GLOBALCONSTANTS DDI (* Global constants *)
  (* Standard: 61499-1 *)
  (* Version 1.0, 2024-02-25, franz *)
  VAR_GLOBAL CONSTANT
    DDI_INTERNAL_DATA_BASE_DDI : UINT := 0; (* 0 - Internal Data Base DDI *)
    DDI_SETPOINT_VOLUME_PER_AREA_APPLICATION_RATE : UINT := 1; (* 1 - Setpoint Volume Per Area Application Rate as *)
    DDI_ACTUAL_VOLUME_PER_AREA_APPLICATION_RATE : UINT := 2; (* 2 - Actual Volume Per Area Application Rate as *)
    DDI_DEFAULT_VOLUME_PER_AREA_APPLICATION_RATE : UINT := 3; (* 3 - Default Volume Per Area Application Rate as *)
    DDI_MINIMUM_VOLUME_PER_AREA_APPLICATION_RATE : UINT := 4; (* 4 - Minimum Volume Per Area Application Rate as *)
    DDI_MAXIMUM_VOLUME_PER_AREA_APPLICATION_RATE : UINT := 5; (* 5 - Maximum Volume Per Area Application Rate as *)
    DDI_SETPOINT_MASS_PER_AREA_APPLICATION_RATE : UINT := 6; (* 6 - Setpoint Mass Per Area Application Rate *)
    DDI_ACTUAL_MASS_PER_AREA_APPLICATION_RATE : UINT := 7; (* 7 - Actual Mass Per Area Application Rate *)
    DDI_DEFAULT_MASS_PER_AREA_APPLICATION_RATE : UINT := 8; (* 8 - Default Mass Per Area Application Rate *)
    DDI_MINIMUM_MASS_PER_AREA_APPLICATION_RATE : UINT := 9; (* 9 - Minimum Mass Per Area Application Rate *)
    DDI_MAXIMUM_MASS_PER_AREA_APPLICATION_RATE : UINT := 10; (* 10 - Maximum Mass Per Area Application Rate *)
    DDI_SETPOINT_COUNT_PER_AREA_APPLICATION_RATE : UINT := 11; (* 11 - Setpoint Count Per Area Application Rate *)
    DDI_ACTUAL_COUNT_PER_AREA_APPLICATION_RATE : UINT := 12; (* 12 - Actual Count Per Area Application Rate *)
    DDI_DEFAULT_COUNT_PER_AREA_APPLICATION_RATE : UINT := 13; (* 13 - Default Count Per Area Application Rate *)
    DDI_MINIMUM_COUNT_PER_AREA_APPLICATION_RATE : UINT := 14; (* 14 - Minimum Count Per Area Application Rate *)
    DDI_MAXIMUM_COUNT_PER_AREA_APPLICATION_RATE : UINT := 15; (* 15 - Maximum Count Per Area Application Rate *)
    DDI_SETPOINT_SPACING_APPLICATION_RATE : UINT := 16; (* 16 - Setpoint Spacing Application Rate *)
    DDI_ACTUAL_SPACING_APPLICATION_RATE : UINT := 17; (* 17 - Actual Spacing Application Rate *)
    DDI_DEFAULT_SPACING_APPLICATION_RATE : UINT := 18; (* 18 - Default Spacing Application Rate *)
    DDI_MINIMUM_SPACING_APPLICATION_RATE : UINT := 19; (* 19 - Minimum Spacing Application Rate *)
    DDI_MAXIMUM_SPACING_APPLICATION_RATE : UINT := 20; (* 20 - Maximum Spacing Application Rate *)
    DDI_SETPOINT_VOLUME_PER_VOLUME_APPLICATION_RATE : UINT := 21; (* 21 - Setpoint Volume Per Volume Application Rate *)
    DDI_ACTUAL_VOLUME_PER_VOLUME_APPLICATION_RATE : UINT := 22; (* 22 - Actual Volume Per Volume Application Rate *)
    DDI_DEFAULT_VOLUME_PER_VOLUME_APPLICATION_RATE : UINT := 23; (* 23 - Default Volume Per Volume Application Rate *)
    DDI_MINIMUM_VOLUME_PER_VOLUME_APPLICATION_RATE : UINT := 24; (* 24 - Minimum Volume Per Volume Application Rate *)
    DDI_MAXIMUM_VOLUME_PER_VOLUME_APPLICATION_RATE : UINT := 25; (* 25 - Maximum Volume Per Volume Application Rate *)
    DDI_SETPOINT_MASS_PER_MASS_APPLICATION_RATE : UINT := 26; (* 26 - Setpoint Mass Per Mass Application Rate *)
    DDI_ACTUAL_MASS_PER_MASS_APPLICATION_RATE : UINT := 27; (* 27 - Actual Mass Per Mass Application Rate *)
    DDI_DEFAULT_MASS_PER_MASS_APPLICATION_RATE : UINT := 28; (* 28 - Default Mass Per Mass Application Rate *)
    DDI_MINIMUM_MASS_PER_MASS_APPLICATION_RATE : UINT := 29; (* 29 - Minimum Mass Per Mass Application Rate *)
    DDI_MAXIMUMMASS_PER_MASS_APPLICATION_RATE : UINT := 30; (* 30 - MaximumMass Per Mass Application Rate *)
    DDI_SETPOINT_VOLUME_PER_MASS_APPLICATION_RATE : UINT := 31; (* 31 - Setpoint Volume Per Mass Application Rate *)
    DDI_ACTUAL_VOLUME_PER_MASS_APPLICATION_RATE : UINT := 32; (* 32 - Actual Volume Per Mass Application Rate *)
    DDI_DEFAULT_VOLUME_PER_MASS_APPLICATION_RATE : UINT := 33; (* 33 - Default Volume Per Mass Application Rate *)
    DDI_MINIMUM_VOLUME_PER_MASS_APPLICATION_RATE : UINT := 34; (* 34 - Minimum Volume Per Mass Application Rate *)
    DDI_MAXIMUM_VOLUME_PER_MASS_APPLICATION_RATE : UINT := 35; (* 35 - Maximum Volume Per Mass Application Rate *)
    DDI_SETPOINT_VOLUME_PER_TIME_APPLICATION_RATE : UINT := 36; (* 36 - Setpoint Volume Per Time Application Rate *)
    DDI_ACTUAL_VOLUME_PER_TIME_APPLICATION_RATE : UINT := 37; (* 37 - Actual Volume Per Time Application Rate *)
    DDI_DEFAULT_VOLUME_PER_TIME_APPLICATION_RATE : UINT := 38; (* 38 - Default Volume Per Time Application Rate *)
    DDI_MINIMUM_VOLUME_PER_TIME_APPLICATION_RATE : UINT := 39; (* 39 - Minimum Volume Per Time Application Rate *)
    DDI_MAXIMUM_VOLUME_PER_TIME_APPLICATION_RATE : UINT := 40; (* 40 - Maximum Volume Per Time Application Rate *)
    DDI_SETPOINT_MASS_PER_TIME_APPLICATION_RATE : UINT := 41; (* 41 - Setpoint Mass Per Time Application Rate *)
    DDI_ACTUAL_MASS_PER_TIME_APPLICATION_RATE : UINT := 42; (* 42 - Actual Mass Per Time Application Rate *)
    DDI_DEFAULT_MASS_PER_TIME_APPLICATION_RATE : UINT := 43; (* 43 - Default Mass Per Time Application Rate *)
    DDI_MINIMUM_MASS_PER_TIME_APPLICATION_RATE : UINT := 44; (* 44 - Minimum Mass Per Time Application Rate *)
    DDI_MAXIMUM_MASS_PER_TIME_APPLICATION_RATE : UINT := 45; (* 45 - Maximum Mass Per Time Application Rate *)
    DDI_SETPOINT_COUNT_PER_TIME_APPLICATION_RATE : UINT := 46; (* 46 - Setpoint Count Per Time Application Rate *)
    DDI_ACTUAL_COUNT_PER_TIME_APPLICATION_RATE : UINT := 47; (* 47 - Actual Count Per Time Application Rate *)
    DDI_DEFAULT_COUNT_PER_TIME_APPLICATION_RATE : UINT := 48; (* 48 - Default Count Per Time Application Rate *)
    DDI_MINIMUM_COUNT_PER_TIME_APPLICATION_RATE : UINT := 49; (* 49 - Minimum Count Per Time Application Rate *)
    DDI_MAXIMUM_COUNT_PER_TIME_APPLICATION_RATE : UINT := 50; (* 50 - Maximum Count Per Time Application Rate *)
    DDI_SETPOINT_TILLAGE_DEPTH : UINT := 51; (* 51 - Setpoint Tillage Depth *)
    DDI_ACTUAL_TILLAGE_DEPTH : UINT := 52; (* 52 - Actual Tillage Depth *)
    DDI_DEFAULT_TILLAGE_DEPTH : UINT := 53; (* 53 - Default Tillage Depth *)
    DDI_MINIMUM_TILLAGE_DEPTH : UINT := 54; (* 54 - Minimum Tillage Depth *)
    DDI_MAXIMUM_TILLAGE_DEPTH : UINT := 55; (* 55 - Maximum Tillage Depth *)
    DDI_SETPOINT_SEEDING_DEPTH : UINT := 56; (* 56 - Setpoint Seeding Depth *)
    DDI_ACTUAL_SEEDING_DEPTH : UINT := 57; (* 57 - Actual Seeding Depth *)
    DDI_DEFAULT_SEEDING_DEPTH : UINT := 58; (* 58 - Default Seeding Depth *)
    DDI_MINIMUM_SEEDING_DEPTH : UINT := 59; (* 59 - Minimum Seeding Depth *)
    DDI_MAXIMUM_SEEDING_DEPTH : UINT := 60; (* 60 - Maximum Seeding Depth *)
    DDI_SETPOINT_WORKING_HEIGHT : UINT := 61; (* 61 - Setpoint Working Height *)
    DDI_ACTUAL_WORKING_HEIGHT : UINT := 62; (* 62 - Actual Working Height *)
    DDI_DEFAULT_WORKING_HEIGHT : UINT := 63; (* 63 - Default Working Height *)
    DDI_MINIMUM_WORKING_HEIGHT : UINT := 64; (* 64 - Minimum Working Height *)
    DDI_MAXIMUM_WORKING_HEIGHT : UINT := 65; (* 65 - Maximum Working Height *)
    DDI_SETPOINT_WORKING_WIDTH : UINT := 66; (* 66 - Setpoint Working Width *)
    DDI_ACTUAL_WORKING_WIDTH : UINT := 67; (* 67 - Actual Working Width *)
    DDI_DEFAULT_WORKING_WIDTH : UINT := 68; (* 68 - Default Working Width *)
    DDI_MINIMUM_WORKING_WIDTH : UINT := 69; (* 69 - Minimum Working Width *)
    DDI_MAXIMUM_WORKING_WIDTH : UINT := 70; (* 70 - Maximum Working Width *)
    DDI_SETPOINT_VOLUME_CONTENT : UINT := 71; (* 71 - Setpoint Volume Content *)
    DDI_ACTUAL_VOLUME_CONTENT : UINT := 72; (* 72 - Actual Volume Content *)
    DDI_MAXIMUM_VOLUME_CONTENT : UINT := 73; (* 73 - Maximum Volume Content *)
    DDI_SETPOINT_MASS_CONTENT : UINT := 74; (* 74 - Setpoint Mass Content *)
    DDI_ACTUAL_MASS_CONTENT : UINT := 75; (* 75 - Actual Mass Content *)
    DDI_MAXIMUM_MASS_CONTENT : UINT := 76; (* 76 - Maximum Mass Content *)
    DDI_SETPOINT_COUNT_CONTENT : UINT := 77; (* 77 - Setpoint Count Content *)
    DDI_ACTUAL_COUNT_CONTENT : UINT := 78; (* 78 - Actual Count Content *)
    DDI_MAXIMUM_COUNT_CONTENT : UINT := 79; (* 79 - Maximum Count Content *)
    DDI_APPLICATION_TOTAL_VOLUME_AS_L : UINT := 80; (* 80 - Application Total Volume as [L] *)
    DDI_APPLICATION_TOTAL_MASS_IN_KG : UINT := 81; (* 81 - Application Total Mass in [kg] *)
    DDI_APPLICATION_TOTAL_COUNT : UINT := 82; (* 82 - Application Total Count *)
    DDI_VOLUME_PER_AREA_YIELD : UINT := 83; (* 83 - Volume Per Area Yield *)
    DDI_MASS_PER_AREA_YIELD : UINT := 84; (* 84 - Mass Per Area Yield *)
    DDI_COUNT_PER_AREA_YIELD : UINT := 85; (* 85 - Count Per Area Yield *)
    DDI_VOLUME_PER_TIME_YIELD : UINT := 86; (* 86 - Volume Per Time Yield *)
    DDI_MASS_PER_TIME_YIELD : UINT := 87; (* 87 - Mass Per Time Yield *)
    DDI_COUNT_PER_TIME_YIELD : UINT := 88; (* 88 - Count Per Time Yield *)
    DDI_YIELD_TOTAL_VOLUME : UINT := 89; (* 89 - Yield Total Volume *)
    DDI_YIELD_TOTAL_MASS : UINT := 90; (* 90 - Yield Total Mass *)
    DDI_YIELD_TOTAL_COUNT : UINT := 91; (* 91 - Yield Total Count *)
    DDI_VOLUME_PER_AREA_CROP_LOSS : UINT := 92; (* 92 - Volume Per Area Crop Loss *)
    DDI_MASS_PER_AREA_CROP_LOSS : UINT := 93; (* 93 - Mass Per Area Crop Loss *)
    DDI_COUNT_PER_AREA_CROP_LOSS : UINT := 94; (* 94 - Count Per Area Crop Loss *)
    DDI_VOLUME_PER_TIME_CROP_LOSS : UINT := 95; (* 95 - Volume Per Time Crop Loss *)
    DDI_MASS_PER_TIME_CROP_LOSS : UINT := 96; (* 96 - Mass Per Time Crop Loss *)
    DDI_COUNT_PER_TIME_CROP_LOSS : UINT := 97; (* 97 - Count Per Time Crop Loss *)
    DDI_PERCENTAGE_CROP_LOSS : UINT := 98; (* 98 - Percentage Crop Loss *)
    DDI_CROP_MOISTURE : UINT := 99; (* 99 - Crop Moisture *)
    DDI_CROP_CONTAMINATION : UINT := 100; (* 100 - Crop Contamination *)
    DDI_SETPOINT_BALE_WIDTH : UINT := 101; (* 101 - Setpoint Bale Width *)
    DDI_ACTUAL_BALE_WIDTH : UINT := 102; (* 102 - Actual Bale Width *)
    DDI_DEFAULT_BALE_WIDTH : UINT := 103; (* 103 - Default Bale Width *)
    DDI_MINIMUM_BALE_WIDTH : UINT := 104; (* 104 - Minimum Bale Width *)
    DDI_MAXIMUM_BALE_WIDTH : UINT := 105; (* 105 - Maximum Bale Width *)
    DDI_SETPOINT_BALE_HEIGHT : UINT := 106; (* 106 - Setpoint Bale Height *)
    DDI_ACTUALBALEHEIGHT : UINT := 107; (* 107 - ActualBaleHeight *)
    DDI_DEFAULT_BALE_HEIGHT : UINT := 108; (* 108 - Default Bale Height *)
    DDI_MINIMUM_BALE_HEIGHT : UINT := 109; (* 109 - Minimum Bale Height *)
    DDI_MAXIMUM_BALE_HEIGHT : UINT := 110; (* 110 - Maximum Bale Height *)
    DDI_SETPOINT_BALE_SIZE : UINT := 111; (* 111 - Setpoint Bale Size *)
    DDI_ACTUAL_BALE_SIZE : UINT := 112; (* 112 - Actual Bale Size *)
    DDI_DEFAULT_BALE_SIZE : UINT := 113; (* 113 - Default Bale Size *)
    DDI_MINIMUM_BALE_SIZE : UINT := 114; (* 114 - Minimum Bale Size *)
    DDI_MAXIMUM_BALE_SIZE : UINT := 115; (* 115 - Maximum Bale Size *)
    DDI_TOTAL_AREA : UINT := 116; (* 116 - Total Area *)
    DDI_EFFECTIVE_TOTAL_DISTANCE : UINT := 117; (* 117 - Effective Total Distance *)
    DDI_INEFFECTIVE_TOTAL_DISTANCE : UINT := 118; (* 118 - Ineffective Total Distance *)
    DDI_EFFECTIVE_TOTAL_TIME : UINT := 119; (* 119 - Effective Total Time *)
    DDI_INEFFECTIVE_TOTAL_TIME : UINT := 120; (* 120 - Ineffective Total Time *)
    DDI_PRODUCT_DENSITY_MASS_PER_VOLUME : UINT := 121; (* 121 - Product Density Mass Per Volume *)
    DDI_PRODUCT_DENSITY_MASS_PERCOUNT : UINT := 122; (* 122 - Product Density Mass PerCount *)
    DDI_PRODUCT_DENSITY_VOLUME_PER_COUNT : UINT := 123; (* 123 - Product Density Volume Per Count *)
    DDI_AUXILIARY_VALVE_SCALING_EXTEND : UINT := 124; (* 124 - Auxiliary Valve Scaling Extend *)
    DDI_AUXILIARY_VALVE_SCALING_RETRACT : UINT := 125; (* 125 - Auxiliary Valve Scaling Retract *)
    DDI_AUXILIARY_VALVE_RAMP_EXTEND_UP : UINT := 126; (* 126 - Auxiliary Valve Ramp Extend Up *)
    DDI_AUXILIARY_VALVE_RAMP_EXTEND_DOWN : UINT := 127; (* 127 - Auxiliary Valve Ramp Extend Down *)
    DDI_AUXILIARY_VALVE_RAMP_RETRACT_UP : UINT := 128; (* 128 - Auxiliary Valve Ramp Retract Up *)
    DDI_AUXILIARY_VALVE_RAMP_RETRACT_DOWN : UINT := 129; (* 129 - Auxiliary Valve Ramp Retract Down *)
    DDI_AUXILIARY_VALVE_FLOAT_THRESHOLD : UINT := 130; (* 130 - Auxiliary Valve Float Threshold *)
    DDI_AUXILIARY_VALVE_PROGRESSIVITY_EXTEND : UINT := 131; (* 131 - Auxiliary Valve Progressivity Extend *)
    DDI_AUXILIARY_VALVE_PROGRESSIVITY_RETRACT : UINT := 132; (* 132 - Auxiliary Valve Progressivity Retract *)
    DDI_AUXILIARY_VALVE_INVERT_PORTS : UINT := 133; (* 133 - Auxiliary Valve Invert Ports *)
    DDI_DEVICE_ELEMENT_OFFSET_X : UINT := 134; (* 134 - Device Element Offset X *)
    DDI_DEVICE_ELEMENT_OFFSET_Y : UINT := 135; (* 135 - Device Element Offset Y *)
    DDI_DEVICE_ELEMENT_OFFSET_Z : UINT := 136; (* 136 - Device Element Offset Z *)
    DDI_DEVICE_VOLUME_CAPACITY : UINT := 137; (* 137 - Device Volume Capacity *)
    DDI_DEVICE_MASS_CAPACITY : UINT := 138; (* 138 - Device Mass Capacity *)
    DDI_DEVICE_COUNT_CAPACITY : UINT := 139; (* 139 - Device Count Capacity *)
    DDI_SETPOINT_PERCENTAGE_APPLICATION_RATE : UINT := 140; (* 140 - Setpoint Percentage Application Rate *)
    DDI_ACTUAL_WORK_STATE : UINT := 141; (* 141 - Actual Work State *)
    DDI_PHYSICAL_SETPOINT_TIME_LATENCY : UINT := 142; (* 142 - Physical Setpoint Time Latency *)
    DDI_PHYSICAL_ACTUAL_VALUE_TIME_LATENCY : UINT := 143; (* 143 - Physical Actual Value Time Latency *)
    DDI_YAW_ANGLE : UINT := 144; (* 144 - Yaw Angle *)
    DDI_ROLL_ANGLE : UINT := 145; (* 145 - Roll Angle *)
    DDI_PITCH_ANGLE : UINT := 146; (* 146 - Pitch Angle *)
    DDI_LOG_COUNT : UINT := 147; (* 147 - Log Count *)
    DDI_TOTAL_FUEL_CONSUMPTION : UINT := 148; (* 148 - Total Fuel Consumption *)
    DDI_INSTANTANEOUS_FUEL_CONSUMPTION_PER_TIME : UINT := 149; (* 149 - Instantaneous Fuel Consumption per Time *)
    DDI_INSTANTANEOUS_FUEL_CONSUMPTION_PER_AREA : UINT := 150; (* 150 - Instantaneous Fuel Consumption per Area *)
    DDI_INSTANTANEOUS_AREA_PER_TIME_CAPACITY : UINT := 151; (* 151 - Instantaneous Area Per Time Capacity *)
    DDI_ACTUAL_NORMALIZED_DIFFERENCE_VEGETATIVE_INDEX_NDVI : UINT := 153; (* 153 - Actual Normalized Difference *)
    DDI_PHYSICAL_OBJECT_LENGTH : UINT := 154; (* 154 - Physical Object Length *)
    DDI_PHYSICAL_OBJECT_WIDTH : UINT := 155; (* 155 - Physical Object Width *)
    DDI_PHYSICAL_OBJECT_HEIGHT : UINT := 156; (* 156 - Physical Object Height *)
    DDI_CONNECTOR_TYPE : UINT := 157; (* 157 - Connector Type *)
    DDI_PRESCRIPTION_CONTROL_STATE : UINT := 158; (* 158 - Prescription Control State *)
    DDI_NUMBER_OF_SUB_UNITS_PER_SECTION : UINT := 159; (* 159 - Number of Sub-Units per Section *)
    DDI_SECTION_CONTROL_STATE : UINT := 160; (* 160 - Section Control State *)
    DDI_ACTUAL_CONDENSED_WORK_STATE_1_16 : UINT := 161; (* 161 - Actual Condensed Work State (1-16) *)
    DDI_ACTUAL_CONDENSED_WORK_STATE_17_32 : UINT := 162; (* 162 - Actual Condensed Work State (17-32) *)
    DDI_ACTUAL_CONDENSED_WORK_STATE_33_48 : UINT := 163; (* 163 - Actual Condensed Work State (33-48) *)
    DDI_ACTUAL_CONDENSED_WORK_STATE_49_64 : UINT := 164; (* 164 - Actual Condensed Work State (49-64) *)
    DDI_ACTUAL_CONDENSED_WORK_STATE_65_80 : UINT := 165; (* 165 - Actual Condensed Work State (65-80) *)
    DDI_ACTUAL_CONDENSED_WORK_STATE_81_96 : UINT := 166; (* 166 - Actual Condensed Work State (81-96) *)
    DDI_ACTUAL_CONDENSED_WORK_STATE_97_112 : UINT := 167; (* 167 - Actual Condensed Work State (97-112) *)
    DDI_ACTUAL_CONDENSED_WORK_STATE_113_128 : UINT := 168; (* 168 - Actual Condensed Work State (113-128) *)
    DDI_ACTUAL_CONDENSED_WORK_STATE_129_144 : UINT := 169; (* 169 - Actual Condensed Work State (129-144) *)
    DDI_ACTUAL_CONDENSED_WORK_STATE_145_160 : UINT := 170; (* 170 - Actual Condensed Work State (145-160) *)
    DDI_ACTUAL_CONDENSED_WORK_STATE_161_176 : UINT := 171; (* 171 - Actual Condensed Work State (161-176) *)
    DDI_ACTUAL_CONDENSED_WORK_STATE_177_192 : UINT := 172; (* 172 - Actual Condensed Work State (177-192) *)
    DDI_ACTUAL_CONDENSED_WORK_STATE_193_208 : UINT := 173; (* 173 - Actual Condensed Work State (193-208) *)
    DDI_ACTUAL_CONDENSED_WORK_STATE_209_224 : UINT := 174; (* 174 - Actual Condensed Work State (209-224) *)
    DDI_ACTUAL_CONDENSED_WORK_STATE_225_240 : UINT := 175; (* 175 - Actual Condensed Work State (225-240) *)
    DDI_ACTUAL_CONDENSED_WORK_STATE_241_256 : UINT := 176; (* 176 - Actual Condensed Work State (241-256) *)
    DDI_ACTUAL_LENGTH_OF_CUT : UINT := 177; (* 177 - Actual length of cut *)
    DDI_ELEMENT_TYPE_INSTANCE : UINT := 178; (* 178 - Element Type Instance *)
    DDI_ACTUAL_CULTURAL_PRACTICE : UINT := 179; (* 179 - Actual Cultural Practice *)
    DDI_DEVICE_REFERENCE_POINT_DRP_TO_GROUND_DISTANCE : UINT := 180; (* 180 - Device Reference Point (DRP) to *)
    DDI_DRY_MASS_PER_AREA_YIELD : UINT := 181; (* 181 - Dry Mass Per Area Yield *)
    DDI_DRY_MASS_PER_TIME_YIELD : UINT := 182; (* 182 - Dry Mass Per Time Yield *)
    DDI_YIELD_TOTAL_DRY_MASS : UINT := 183; (* 183 - Yield Total Dry Mass *)
    DDI_REFERENCE_MOISTURE_FOR_DRY_MASS : UINT := 184; (* 184 - Reference Moisture For Dry Mass *)
    DDI_SEED_COTTON_MASS_PER_AREA_YIELD : UINT := 185; (* 185 - Seed Cotton Mass Per Area Yield *)
    DDI_LINT_COTTON_MASS_PER_AREA_YIELD : UINT := 186; (* 186 - Lint Cotton Mass Per Area Yield *)
    DDI_SEED_COTTON_MASS_PER_TIME_YIELD : UINT := 187; (* 187 - Seed Cotton Mass Per Time Yield *)
    DDI_LINT_COTTON_MASS_PER_TIME_YIELD : UINT := 188; (* 188 - Lint Cotton Mass Per Time Yield *)
    DDI_YIELD_TOTAL_SEED_COTTON_MASS : UINT := 189; (* 189 - Yield Total Seed Cotton Mass *)
    DDI_YIELD_TOTAL_LINT_COTTON_MASS : UINT := 190; (* 190 - Yield Total Lint Cotton Mass *)
    DDI_LINT_TURNOUT_PERCENTAGE : UINT := 191; (* 191 - Lint Turnout Percentage *)
    DDI_AMBIENT_TEMPERATURE : UINT := 192; (* 192 - Ambient temperature *)
    DDI_SETPOINT_PRODUCT_PRESSURE : UINT := 193; (* 193 - Setpoint Product Pressure *)
    DDI_ACTUAL_PRODUCT_PRESSURE : UINT := 194; (* 194 - Actual Product Pressure *)
    DDI_MINIMUM_PRODUCT_PRESSURE : UINT := 195; (* 195 - Minimum Product Pressure *)
    DDI_MAXIMUM_PRODUCT_PRESSURE : UINT := 196; (* 196 - Maximum Product Pressure *)
    DDI_SETPOINT_PUMP_OUTPUT_PRESSURE : UINT := 197; (* 197 - Setpoint Pump Output Pressure *)
    DDI_ACTUAL_PUMP_OUTPUT_PRESSURE : UINT := 198; (* 198 - Actual Pump Output Pressure *)
    DDI_MINIMUM_PUMP_OUTPUT_PRESSURE : UINT := 199; (* 199 - Minimum Pump Output Pressure *)
    DDI_MAXIMUM_PUMP_OUTPUT_PRESSURE : UINT := 200; (* 200 - Maximum Pump Output Pressure *)
    DDI_SETPOINT_TANK_AGITATION_PRESSURE : UINT := 201; (* 201 - Setpoint Tank Agitation Pressure *)
    DDI_ACTUAL_TANK_AGITATION_PRESSURE : UINT := 202; (* 202 - Actual Tank Agitation Pressure *)
    DDI_MINIMUM_TANK_AGITATION_PRESSURE : UINT := 203; (* 203 - Minimum Tank Agitation Pressure *)
    DDI_MAXIMUM_TANK_AGITATION_PRESSURE : UINT := 204; (* 204 - Maximum Tank Agitation Pressure *)
    DDI_SC_SETPOINT_TURN_ON_TIME : UINT := 205; (* 205 - SC Setpoint Turn On Time *)
    DDI_SC_SETPOINT_TURN_OFF_TIME : UINT := 206; (* 206 - SC Setpoint Turn Off Time *)
    DDI_WIND_SPEED : UINT := 207; (* 207 - Wind speed *)
    DDI_WIND_DIRECTION : UINT := 208; (* 208 - Wind direction *)
    DDI_RELATIVE_HUMIDITY : UINT := 209; (* 209 - Relative Humidity *)
    DDI_SKY_CONDITIONS : UINT := 210; (* 210 - Sky conditions *)
    DDI_LAST_BALE_FLAKES_PER_BALE : UINT := 211; (* 211 - Last Bale Flakes per Bale *)
    DDI_LAST_BALE_AVERAGE_MOISTURE : UINT := 212; (* 212 - Last Bale Average Moisture *)
    DDI_LAST_BALE_AVERAGE_STROKES_PER_FLAKE : UINT := 213; (* 213 - Last Bale Average Strokes per Flake *)
    DDI_LIFETIME_BALE_COUNT : UINT := 214; (* 214 - Lifetime Bale Count *)
    DDI_LIFETIME_WORKING_HOURS : UINT := 215; (* 215 - Lifetime Working Hours *)
    DDI_ACTUAL_BALE_HYDRAULIC_PRESSURE : UINT := 216; (* 216 - Actual Bale Hydraulic Pressure *)
    DDI_LAST_BALE_AVERAGE_HYDRAULIC_PRESSURE : UINT := 217; (* 217 - Last Bale Average Hydraulic Pressure *)
    DDI_SETPOINT_BALE_COMPRESSION_PLUNGER_LOAD : UINT := 218; (* 218 - Setpoint Bale Compression Plunger Load *)
    DDI_ACTUAL_BALE_COMPRESSION_PLUNGER_LOAD : UINT := 219; (* 219 - Actual Bale Compression Plunger Load *)
    DDI_LAST_BALE_AVERAGE_BALE_COMPRESSION_PLUNGER_LOAD : UINT := 220; (* 220 - Last Bale Average Bale Compression *)
    DDI_LAST_BALE_APPLIED_PRESERVATIVE : UINT := 221; (* 221 - Last Bale Applied Preservative *)
    DDI_LAST_BALE_TAG_NUMBER : UINT := 222; (* 222 - Last Bale Tag Number *)
    DDI_LAST_BALE_MASS : UINT := 223; (* 223 - Last Bale Mass *)
    DDI_DELTA_T : UINT := 224; (* 224 - Delta T *)
    DDI_SETPOINT_WORKING_LENGTH : UINT := 225; (* 225 - Setpoint Working Length *)
    DDI_ACTUAL_WORKING_LENGTH : UINT := 226; (* 226 - Actual Working Length *)
    DDI_MINIMUM_WORKING_LENGTH : UINT := 227; (* 227 - Minimum Working Length *)
    DDI_MAXIMUM_WORKING_LENGTH : UINT := 228; (* 228 - Maximum Working Length *)
    DDI_ACTUAL_NET_WEIGHT : UINT := 229; (* 229 - Actual Net Weight *)
    DDI_NET_WEIGHT_STATE : UINT := 230; (* 230 - Net Weight State *)
    DDI_SETPOINT_NET_WEIGHT : UINT := 231; (* 231 - Setpoint Net Weight *)
    DDI_ACTUAL_GROSS_WEIGHT : UINT := 232; (* 232 - Actual Gross Weight *)
    DDI_GROSS_WEIGHT_STATE : UINT := 233; (* 233 - Gross Weight State *)
    DDI_MINIMUM_GROSS_WEIGHT : UINT := 234; (* 234 - Minimum Gross Weight *)
    DDI_MAXIMUM_GROSS_WEIGHT : UINT := 235; (* 235 - Maximum Gross Weight *)
    DDI_THRESHER_ENGAGEMENT_TOTAL_TIME : UINT := 236; (* 236 - Thresher Engagement Total Time *)
    DDI_ACTUAL_HEADER_WORKING_HEIGHT_STATUS : UINT := 237; (* 237 - Actual Header Working Height Status *)
    DDI_ACTUAL_HEADER_ROTATIONAL_SPEED_STATUS : UINT := 238; (* 238 - Actual Header Rotational Speed Status *)
    DDI_YIELD_HOLD_STATUS : UINT := 239; (* 239 - Yield Hold Status *)
    DDI_ACTUAL_UNLOADING_SYSTEM_STATUS : UINT := 240; (* 240 - Actual (Un)Loading System Status *)
    DDI_CROP_TEMPERATURE : UINT := 241; (* 241 - Crop Temperature *)
    DDI_SETPOINT_SIEVE_CLEARANCE : UINT := 242; (* 242 - Setpoint Sieve Clearance *)
    DDI_ACTUAL_SIEVE_CLEARANCE : UINT := 243; (* 243 - Actual Sieve Clearance *)
    DDI_MINIMUM_SIEVE_CLEARANCE : UINT := 244; (* 244 - Minimum Sieve Clearance *)
    DDI_MAXIMUM_SIEVE_CLEARANCE : UINT := 245; (* 245 - Maximum Sieve Clearance *)
    DDI_SETPOINT_CHAFFER_CLEARANCE : UINT := 246; (* 246 - Setpoint Chaffer Clearance *)
    DDI_ACTUAL_CHAFFER_CLEARANCE : UINT := 247; (* 247 - Actual Chaffer Clearance *)
    DDI_MINIMUM_CHAFFER_CLEARANCE : UINT := 248; (* 248 - Minimum Chaffer Clearance *)
    DDI_MAXIMUM_CHAFFER_CLEARANCE : UINT := 249; (* 249 - Maximum Chaffer Clearance *)
    DDI_SETPOINT_CONCAVE_CLEARANCE : UINT := 250; (* 250 - Setpoint Concave Clearance *)
    DDI_ACTUAL_CONCAVE_CLEARANCE : UINT := 251; (* 251 - Actual Concave Clearance *)
    DDI_MINIMUM_CONCAVE_CLEARANCE : UINT := 252; (* 252 - Minimum Concave Clearance *)
    DDI_MAXIMUM_CONCAVE_CLEARANCE : UINT := 253; (* 253 - Maximum Concave Clearance *)
    DDI_SETPOINT_SEPARATION_FAN_ROTATIONAL_SPEED : UINT := 254; (* 254 - Setpoint Separation Fan Rotational Speed *)
    DDI_ACTUAL_SEPARATION_FAN_ROTATIONAL_SPEED : UINT := 255; (* 255 - Actual Separation Fan Rotational Speed *)
    DDI_MINIMUM_SEPARATION_FAN_ROTATIONAL_SPEED : UINT := 256; (* 256 - Minimum Separation Fan Rotational Speed *)
    DDI_MAXIMUM_SEPARATION_FAN_ROTATIONAL_SPEED : UINT := 257; (* 257 - Maximum Separation Fan Rotational Speed *)
    DDI_HYDRAULIC_OIL_TEMPERATURE : UINT := 258; (* 258 - Hydraulic Oil Temperature *)
    DDI_YIELD_LAG_IGNORE_TIME : UINT := 259; (* 259 - Yield Lag Ignore Time *)
    DDI_YIELD_LEAD_IGNORE_TIME : UINT := 260; (* 260 - Yield Lead Ignore Time *)
    DDI_AVERAGE_YIELD_MASS_PER_TIME : UINT := 261; (* 261 - Average Yield Mass Per Time *)
    DDI_AVERAGE_CROP_MOISTURE : UINT := 262; (* 262 - Average Crop Moisture *)
    DDI_AVERAGE_YIELD_MASS_PER_AREA : UINT := 263; (* 263 - Average Yield Mass Per Area *)
    DDI_CONNECTOR_PIVOT_X_OFFSET : UINT := 264; (* 264 - Connector Pivot X-Offset *)
    DDI_REMAINING_AREA : UINT := 265; (* 265 - Remaining Area *)
    DDI_LIFETIME_APPLICATION_TOTAL_MASS : UINT := 266; (* 266 - Lifetime Application Total Mass *)
    DDI_LIFETIME_APPLICATION_TOTAL_COUNT : UINT := 267; (* 267 - Lifetime Application Total Count *)
    DDI_LIFETIME_YIELD_TOTAL_VOLUME : UINT := 268; (* 268 - Lifetime Yield Total Volume *)
    DDI_LIFETIME_YIELD_TOTAL_MASS : UINT := 269; (* 269 - Lifetime Yield Total Mass *)
    DDI_LIFETIME_YIELD_TOTAL_COUNT : UINT := 270; (* 270 - Lifetime Yield Total Count *)
    DDI_LIFETIME_TOTAL_AREA : UINT := 271; (* 271 - Lifetime Total Area *)
    DDI_LIFETIME_EFFECTIVE_TOTAL_DISTANCE : UINT := 272; (* 272 - Lifetime Effective Total Distance *)
    DDI_LIFETIME_INEFFECTIVE_TOTAL_DISTANCE : UINT := 273; (* 273 - Lifetime Ineffective Total Distance *)
    DDI_LIFETIME_EFFECTIVE_TOTAL_TIME : UINT := 274; (* 274 - Lifetime Effective Total Time *)
    DDI_LIFETIME_INEFFECTIVE_TOTAL_TIME : UINT := 275; (* 275 - Lifetime Ineffective Total Time *)
    DDI_LIFETIME_FUEL_CONSUMPTION : UINT := 276; (* 276 - Lifetime Fuel Consumption *)
    DDI_LIFETIME_AVERAGE_FUEL_CONSUMPTION_PER_TIME : UINT := 277; (* 277 - Lifetime Average Fuel Consumption per Time *)
    DDI_LIFETIME_AVERAGE_FUEL_CONSUMPTION_PER_AREA : UINT := 278; (* 278 - Lifetime Average Fuel Consumption per Area *)
    DDI_LIFETIME_YIELD_TOTAL_DRY_MASS : UINT := 279; (* 279 - Lifetime Yield Total Dry Mass *)
    DDI_LIFETIME_YIELD_TOTAL_SEED_COTTON_MASS : UINT := 280; (* 280 - Lifetime Yield Total Seed Cotton Mass *)
    DDI_LIFETIME_YIELD_TOTAL_LINT_COTTON_MASS : UINT := 281; (* 281 - Lifetime Yield Total Lint Cotton Mass *)
    DDI_LIFETIME_THRESHING_ENGAGEMENT_TOTAL_TIME : UINT := 282; (* 282 - Lifetime Threshing Engagement Total Time *)
    DDI_PRECUT_TOTAL_COUNT : UINT := 283; (* 283 - Precut Total Count *)
    DDI_UNCUT_TOTAL_COUNT : UINT := 284; (* 284 - Uncut Total Count *)
    DDI_LIFETIME_PRECUT_TOTAL_COUNT : UINT := 285; (* 285 - Lifetime Precut Total Count *)
    DDI_LIFETIME_UNCUT_TOTAL_COUNT : UINT := 286; (* 286 - Lifetime Uncut Total Count *)
    DDI_SETPOINT_PRESCRIPTION_MODE : UINT := 287; (* 287 - Setpoint Prescription Mode *)
    DDI_ACTUAL_PRESCRIPTION_MODE : UINT := 288; (* 288 - Actual Prescription Mode *)
    DDI_SETPOINT_WORK_STATE : UINT := 289; (* 289 - Setpoint Work State *)
    DDI_SETPOINT_CONDENSED_WORK_STATE_1_16 : UINT := 290; (* 290 - Setpoint Condensed Work State (1-16) *)
    DDI_SETPOINT_CONDENSED_WORK_STATE_17_32 : UINT := 291; (* 291 - Setpoint Condensed Work State (17-32) *)
    DDI_SETPOINT_CONDENSED_WORK_STATE_33_48 : UINT := 292; (* 292 - Setpoint Condensed Work State (33-48) *)
    DDI_SETPOINT_CONDENSED_WORK_STATE_49_64 : UINT := 293; (* 293 - Setpoint Condensed Work State (49-64) *)
    DDI_SETPOINT_CONDENSED_WORK_STATE_65_80 : UINT := 294; (* 294 - Setpoint Condensed Work State (65-80) *)
    DDI_SETPOINT_CONDENSED_WORK_STATE_81_96 : UINT := 295; (* 295 - Setpoint Condensed Work State (81-96) *)
    DDI_SETPOINT_CONDENSED_WORK_STATE_97_112 : UINT := 296; (* 296 - Setpoint Condensed Work State (97-112) *)
    DDI_SETPOINT_CONDENSED_WORK_STATE_113_128 : UINT := 297; (* 297 - Setpoint Condensed Work State (113-128) *)
    DDI_SETPOINT_CONDENSED_WORK_STATE_129_144 : UINT := 298; (* 298 - Setpoint Condensed Work State (129-144) *)
    DDI_SETPOINT_CONDENSED_WORK_STATE_145_160 : UINT := 299; (* 299 - Setpoint Condensed Work State (145-160) *)
    DDI_SETPOINT_CONDENSED_WORK_STATE_161_176 : UINT := 300; (* 300 - Setpoint Condensed Work State (161-176) *)
    DDI_SETPOINT_CONDENSED_WORK_STATE_177_192 : UINT := 301; (* 301 - Setpoint Condensed Work State (177-192) *)
    DDI_SETPOINT_CONDENSED_WORK_STATE_193_208 : UINT := 302; (* 302 - Setpoint Condensed Work State (193-208) *)
    DDI_SETPOINT_CONDENSED_WORK_STATE_209_224 : UINT := 303; (* 303 - Setpoint Condensed Work State (209-224) *)
    DDI_SETPOINT_CONDENSED_WORK_STATE_225_240 : UINT := 304; (* 304 - Setpoint Condensed Work State (225-240) *)
    DDI_SETPOINT_CONDENSED_WORK_STATE_241_256 : UINT := 305; (* 305 - Setpoint Condensed Work State (241-256) *)
    DDI_TRUE_ROTATION_POINT_X_OFFSET : UINT := 306; (* 306 - True Rotation Point X-Offset *)
    DDI_TRUE_ROTATION_POINT_Y_OFFSET : UINT := 307; (* 307 - True Rotation Point Y-Offset *)
    DDI_ACTUAL_PERCENTAGE_APPLICATION_RATE : UINT := 308; (* 308 - Actual Percentage Application Rate *)
    DDI_MINIMUM_PERCENTAGE_APPLICATION_RATE : UINT := 309; (* 309 - Minimum Percentage Application Rate *)
    DDI_MAXIMUM_PERCENTAGE_APPLICATION_RATE : UINT := 310; (* 310 - Maximum Percentage Application Rate *)
    DDI_RELATIVE_YIELD_POTENTIAL : UINT := 311; (* 311 - Relative Yield Potential *)
    DDI_MINIMUM_RELATIVE_YIELD_POTENTIAL : UINT := 312; (* 312 - Minimum Relative Yield Potential *)
    DDI_MAXIMUM_RELATIVE_YIELD_POTENTIAL : UINT := 313; (* 313 - Maximum Relative Yield Potential *)
    DDI_ACTUAL_PERCENTAGE_CROP_DRY_MATTER : UINT := 314; (* 314 - Actual Percentage Crop Dry Matter *)
    DDI_AVERAGE_PERCENTAGE_CROP_DRY_MATTER : UINT := 315; (* 315 - Average Percentage Crop Dry Matter *)
    DDI_EFFECTIVE_TOTAL_FUEL_CONSUMPTION : UINT := 316; (* 316 - Effective Total Fuel Consumption *)
    DDI_INEFFECTIVE_TOTAL_FUEL_CONSUMPTION : UINT := 317; (* 317 - Ineffective Total Fuel Consumption *)
    DDI_EFFECTIVE_TOTAL_DIESEL_EXHAUST_FLUID_CONSUMPTION : UINT := 318; (* 318 - Effective Total Diesel Exhaust Fluid *)
    DDI_INEFFECTIVE_TOTAL_DIESEL_EXHAUST_FLUID_CONSUMPTION : UINT := 319; (* 319 - Ineffective Total Diesel Exhaust *)
    DDI_LAST_LOADED_WEIGHT : UINT := 320; (* 320 - Last loaded Weight *)
    DDI_LAST_UNLOADED_WEIGHT : UINT := 321; (* 321 - Last unloaded Weight *)
    DDI_LOAD_IDENTIFICATION_NUMBER : UINT := 322; (* 322 - Load Identification Number *)
    DDI_UNLOAD_IDENTIFICATION_NUMBER : UINT := 323; (* 323 - Unload Identification Number *)
    DDI_CHOPPER_ENGAGEMENT_TOTAL_TIME : UINT := 324; (* 324 - Chopper Engagement Total Time *)
    DDI_LIFETIME_APPLICATION_TOTAL_VOLUME : UINT := 325; (* 325 - Lifetime Application Total Volume *)
    DDI_SETPOINT_HEADER_SPEED : UINT := 326; (* 326 - Setpoint Header Speed *)
    DDI_ACTUAL_HEADER_SPEED : UINT := 327; (* 327 - Actual Header Speed *)
    DDI_MINIMUM_HEADER_SPEED : UINT := 328; (* 328 - Minimum Header Speed *)
    DDI_MAXIMUM_HEADER_SPEED : UINT := 329; (* 329 - Maximum Header Speed *)
    DDI_SETPOINT_CUTTING_DRUM_SPEED : UINT := 330; (* 330 - Setpoint Cutting drum speed *)
    DDI_ACTUAL_CUTTING_DRUM_SPEED : UINT := 331; (* 331 - Actual Cutting drum speed *)
    DDI_MINIMUM_CUTTING_DRUM_SPEED : UINT := 332; (* 332 - Minimum Cutting drum speed *)
    DDI_MAXIMUM_CUTTING_DRUM_SPEED : UINT := 333; (* 333 - Maximum Cutting drum speed *)
    DDI_OPERATING_HOURS_SINCE_LAST_SHARPENING : UINT := 334; (* 334 - Operating Hours Since Last Sharpening *)
    DDI_FRONT_PTO_HOURS : UINT := 335; (* 335 - Front PTO hours *)
    DDI_REAR_PTO_HOURS : UINT := 336; (* 336 - Rear PTO hours *)
    DDI_LIFETIME_FRONT_PTO_HOURS : UINT := 337; (* 337 - Lifetime Front PTO hours *)
    DDI_LIFETIME_REAR_PTO_HOURS : UINT := 338; (* 338 - Lifetime Rear PTO Hours *)
    DDI_EFFECTIVE_TOTAL_LOADING_TIME : UINT := 339; (* 339 - Effective Total Loading Time *)
    DDI_EFFECTIVE_TOTAL_UNLOADING_TIME : UINT := 340; (* 340 - Effective Total Unloading Time *)
    DDI_SETPOINT_GRAIN_KERNEL_CRACKER_GAP : UINT := 341; (* 341 - Setpoint Grain Kernel Cracker Gap *)
    DDI_ACTUAL_GRAIN_KERNEL_CRACKER_GAP : UINT := 342; (* 342 - Actual Grain Kernel Cracker Gap *)
    DDI_MINIMUM_GRAIN_KERNEL_CRACKER_GAP : UINT := 343; (* 343 - Minimum Grain Kernel Cracker Gap *)
    DDI_MAXIMUM_GRAIN_KERNEL_CRACKER_GAP : UINT := 344; (* 344 - Maximum Grain Kernel Cracker Gap *)
    DDI_SETPOINT_SWATHING_WIDTH : UINT := 345; (* 345 - Setpoint Swathing Width *)
    DDI_ACTUAL_SWATHING_WIDTH : UINT := 346; (* 346 - Actual Swathing Width *)
    DDI_MINIMUM_SWATHING_WIDTH : UINT := 347; (* 347 - Minimum Swathing Width *)
    DDI_MAXIMUM_SWATHING_WIDTH : UINT := 348; (* 348 - Maximum Swathing Width *)
    DDI_NOZZLE_DRIFT_REDUCTION : UINT := 349; (* 349 - Nozzle Drift Reduction *)
    DDI_FUNCTION_OR_OPERATION_TECHNIQUE : UINT := 350; (* 350 - Function or Operation Technique *)
    DDI_APPLICATION_TOTAL_VOLUME_IN_ML : UINT := 351; (* 351 - Application Total Volume in [ml] *)
    DDI_APPLICATION_TOTAL_MASS_IN_GRAM_G : UINT := 352; (* 352 - Application Total Mass in gram [g] *)
    DDI_TOTAL_APPLICATION_OF_NITROGEN : UINT := 353; (* 353 - Total Application of Nitrogen *)
    DDI_TOTAL_APPLICATION_OF_AMMONIUM : UINT := 354; (* 354 - Total Application of Ammonium *)
    DDI_TOTAL_APPLICATION_OF_PHOSPHOR : UINT := 355; (* 355 - Total Application of Phosphor *)
    DDI_TOTAL_APPLICATION_OF_POTASSIUM : UINT := 356; (* 356 - Total Application of Potassium *)
    DDI_TOTAL_APPLICATION_OF_DRY_MATTER : UINT := 357; (* 357 - Total Application of Dry Matter *)
    DDI_AVERAGE_DRY_YIELD_MASS_PER_TIME : UINT := 358; (* 358 - Average Dry Yield Mass Per Time *)
    DDI_AVERAGE_DRY_YIELD_MASS_PER_AREA : UINT := 359; (* 359 - Average Dry Yield Mass Per Area *)
    DDI_LAST_BALE_SIZE : UINT := 360; (* 360 - Last Bale Size *)
    DDI_LAST_BALE_DENSITY : UINT := 361; (* 361 - Last Bale Density *)
    DDI_TOTAL_BALE_LENGTH : UINT := 362; (* 362 - Total Bale Length *)
    DDI_LAST_BALE_DRY_MASS : UINT := 363; (* 363 - Last Bale Dry Mass *)
    DDI_ACTUAL_FLAKE_SIZE : UINT := 364; (* 364 - Actual Flake Size *)
    DDI_SETPOINT_DOWNFORCE_PRESSURE : UINT := 365; (* 365 - Setpoint Downforce Pressure *)
    DDI_ACTUAL_DOWNFORCE_PRESSURE : UINT := 366; (* 366 - Actual Downforce Pressure *)
    DDI_CONDENSED_SECTION_OVERRIDE_STATE_1_16 : UINT := 367; (* 367 - Condensed Section Override State (1-16) *)
    DDI_CONDENSED_SECTION_OVERRIDE_STATE_17_32 : UINT := 368; (* 368 - Condensed Section Override State (17-32) *)
    DDI_CONDENSED_SECTION_OVERRIDE_STATE_33_48 : UINT := 369; (* 369 - Condensed Section Override State (33-48) *)
    DDI_CONDENSED_SECTION_OVERRIDE_STATE_49_64 : UINT := 370; (* 370 - Condensed Section Override State (49-64) *)
    DDI_CONDENSED_SECTION_OVERRIDE_STATE_65_80 : UINT := 371; (* 371 - Condensed Section Override State (65-80) *)
    DDI_CONDENSED_SECTION_OVERRIDE_STATE_81_96 : UINT := 372; (* 372 - Condensed Section Override State (81-96) *)
    DDI_CONDENSED_SECTION_OVERRIDE_STATE_97_112 : UINT := 373; (* 373 - Condensed Section Override State (97-112) *)
    DDI_CONDENSED_SECTION_OVERRIDE_STATE_113_128 : UINT := 374; (* 374 - Condensed Section Override State (113-128) *)
    DDI_CONDENSED_SECTION_OVERRIDE_STATE_129_144 : UINT := 375; (* 375 - Condensed Section Override State (129-144) *)
    DDI_CONDENSED_SECTION_OVERRIDE_STATE_145_160 : UINT := 376; (* 376 - Condensed Section Override State (145-160) *)
    DDI_CONDENSED_SECTION_OVERRIDE_STATE_161_176 : UINT := 377; (* 377 - Condensed Section Override State (161-176) *)
    DDI_CONDENSED_SECTION_OVERRIDE_STATE_177_192 : UINT := 378; (* 378 - Condensed Section Override State (177-192) *)
    DDI_CONDENSED_SECTION_OVERRIDE_STATE_193_208 : UINT := 379; (* 379 - Condensed Section Override State (193-208) *)
    DDI_CONDENSED_SECTION_OVERRIDE_STATE_209_224 : UINT := 380; (* 380 - Condensed Section Override State (209-224) *)
    DDI_CONDENSED_SECTION_OVERRIDE_STATE_225_240 : UINT := 381; (* 381 - Condensed Section Override State (225-240) *)
    DDI_CONDENSED_SECTION_OVERRIDE_STATE_241_256 : UINT := 382; (* 382 - Condensed Section Override State (241-256) *)
    DDI_APPARENT_WIND_DIRECTION : UINT := 383; (* 383 - Apparent Wind Direction *)
    DDI_APPARENT_WIND_SPEED : UINT := 384; (* 384 - Apparent Wind Speed *)
    DDI_MSL_ATMOSPHERIC_PRESSURE : UINT := 385; (* 385 - MSL Atmospheric Pressure *)
    DDI_ACTUAL_ATMOSPHERIC_PRESSURE : UINT := 386; (* 386 - Actual Atmospheric Pressure *)
    DDI_TOTAL_REVOLUTIONS_IN_FRACTIONAL_REVOLUTIONS : UINT := 387; (* 387 - Total Revolutions in Fractional *)
    DDI_TOTAL_REVOLUTIONS_IN_COMPLETE_REVOLUTIONS : UINT := 388; (* 388 - Total Revolutions in Complete Revolutions *)
    DDI_SETPOINT_REVOLUTIONS_SPECIFIED_AS_COUNT_PER_TIME : UINT := 389; (* 389 - Setpoint Revolutions specified as *)
    DDI_ACTUAL_REVOLUTIONS_PER_TIME : UINT := 390; (* 390 - Actual Revolutions Per Time *)
    DDI_DEFAULT_REVOLUTIONS_PER_TIME : UINT := 391; (* 391 - Default Revolutions Per Time *)
    DDI_MINIMUM_REVOLUTIONS_PER_TIME : UINT := 392; (* 392 - Minimum Revolutions Per Time *)
    DDI_MAXIMUM_REVOLUTIONS_PER_TIME : UINT := 393; (* 393 - Maximum Revolutions Per Time *)
    DDI_ACTUAL_FUEL_TANK_CONTENT : UINT := 394; (* 394 - Actual Fuel Tank Content *)
    DDI_ACTUAL_DIESEL_EXHAUST_FLUID_TANK_CONTENT : UINT := 395; (* 395 - Actual Diesel Exhaust Fluid Tank Content *)
    DDI_SETPOINT_SPEED : UINT := 396; (* 396 - Setpoint Speed *)
    DDI_ACTUAL_SPEED : UINT := 397; (* 397 - Actual Speed *)
    DDI_MINIMUM_SPEED : UINT := 398; (* 398 - Minimum Speed *)
    DDI_MAXIMUM_SPEED : UINT := 399; (* 399 - Maximum Speed *)
    DDI_SPEED_SOURCE : UINT := 400; (* 400 - Speed Source *)
    DDI_ACTUAL_APPLICATION_OF_NITROGEN : UINT := 401; (* 401 - Actual Application of Nitrogen as [mg/l] *)
    DDI_ACTUAL_APPLICATION_OF_AMMONIUM : UINT := 402; (* 402 - Actual application of Ammonium *)
    DDI_ACTUAL_APPLICATION_OF_PHOSPHOR : UINT := 403; (* 403 - Actual application of Phosphor *)
    DDI_ACTUAL_APPLICATION_OF_POTASSIUM : UINT := 404; (* 404 - Actual application of Potassium *)
    DDI_ACTUAL_APPLICATION_OF_DRY_MATTER : UINT := 405; (* 405 - Actual application of Dry Matter *)
    DDI_ACTUAL_PROTEIN_CONTENT : UINT := 406; (* 406 - Actual Protein Content *)
    DDI_AVERAGE_PROTEIN_CONTENT : UINT := 407; (* 407 - Average Protein Content *)
    DDI_AVERAGE_CROP_CONTAMINATION : UINT := 408; (* 408 - Average Crop Contamination *)
    DDI_TOTAL_DIESEL_EXHAUST_FLUID_CONSUMPTION : UINT := 409; (* 409 - Total Diesel Exhaust Fluid Consumption *)
    DDI_INSTANTANEOUS_DIESEL_EXHAUST_FLUID_CONSUMPTION_PER_TIME : UINT := 410; (* 410 - Instantaneous Diesel Exhaust *)
    DDI_INSTANTANEOUS_DIESEL_EXHAUST_FLUID_CONSUMPTION_PER_AREA : UINT := 411; (* 411 - Instantaneous Diesel Exhaust *)
    DDI_LIFETIME_DIESEL_EXHAUST_FLUID_CONSUMPTION : UINT := 412; (* 412 - Lifetime Diesel Exhaust Fluid Consumption *)
    DDI_LIFETIME_AVERAGE_DIESEL_EXHAUST_FLUID_CONSUMPTION_PER_TIME : UINT := 413; (* 413 - Lifetime Average Diesel *)
    DDI_LIFETIME_AVERAGE_DIESEL_EXHAUST_FLUID_CONSUMPTION_PER_AREA : UINT := 414; (* 414 - Lifetime Average Diesel *)
    DDI_ACTUAL_SEED_SINGULATION_PERCENTAGE : UINT := 415; (* 415 - Actual Seed Singulation Percentage *)
    DDI_AVERAGE_SEED_SINGULATION_PERCENTAGE : UINT := 416; (* 416 - Average Seed Singulation Percentage *)
    DDI_ACTUAL_SEED_SKIP_PERCENTAGE : UINT := 417; (* 417 - Actual Seed Skip Percentage *)
    DDI_AVERAGE_SEED_SKIP_PERCENTAGE : UINT := 418; (* 418 - Average Seed Skip Percentage *)
    DDI_ACTUAL_SEED_MULTIPLE_PERCENTAGE : UINT := 419; (* 419 - Actual Seed Multiple Percentage *)
    DDI_AVERAGE_SEED_MULTIPLE_PERCENTAGE : UINT := 420; (* 420 - Average Seed Multiple Percentage *)
    DDI_ACTUAL_SEED_SPACING_DEVIATION : UINT := 421; (* 421 - Actual Seed Spacing Deviation *)
    DDI_AVERAGE_SEED_SPACING_DEVIATION : UINT := 422; (* 422 - Average Seed Spacing Deviation *)
    DDI_ACTUAL_COEFFICIENT_OF_VARIATION_OF_SEED_SPACING_PERCENTAGE : UINT := 423; (* 423 - Actual Coefficient of *)
    DDI_AVERAGE_COEFFICIENT_OF_VARIATION_OF_SEED_SPACING_PERCENTAGE : UINT := 424; (* 424 - Average Coefficient of *)
    DDI_SETPOINT_MAXIMUM_ALLOWED_SEED_SPACING_DEVIATION : UINT := 425; (* 425 - Setpoint Maximum Allowed Seed Spacing *)
    DDI_SETPOINT_DOWNFORCE_AS_FORCE : UINT := 426; (* 426 - Setpoint Downforce as Force *)
    DDI_ACTUAL_DOWNFORCE_AS_FORCE : UINT := 427; (* 427 - Actual Downforce as Force *)
    DDI_LOADED_TOTAL_MASS : UINT := 428; (* 428 - Loaded Total Mass *)
    DDI_UNLOADED_TOTAL_MASS : UINT := 429; (* 429 - Unloaded Total Mass *)
    DDI_LIFETIME_LOADED_TOTAL_MASS : UINT := 430; (* 430 - Lifetime Loaded Total Mass *)
    DDI_LIFETIME_UNLOADED_TOTAL_MASS : UINT := 431; (* 431 - Lifetime Unloaded Total Mass *)
    DDI_SETPOINT_APPLICATION_RATE_OF_NITROGEN : UINT := 432; (* 432 - Setpoint Application Rate of Nitrogen *)
    DDI_ACTUAL_APPLICATION_RATE_OF_NITROGEN : UINT := 433; (* 433 - Actual Application Rate of Nitrogen *)
    DDI_MINIMUM_APPLICATION_RATE_OF_NITROGEN : UINT := 434; (* 434 - Minimum Application Rate of Nitrogen *)
    DDI_MAXIMUM_APPLICATION_RATE_OF_NITROGEN : UINT := 435; (* 435 - Maximum Application Rate of Nitrogen *)
    DDI_SETPOINT_APPLICATION_RATE_OF_AMMONIUM : UINT := 436; (* 436 - Setpoint Application Rate of Ammonium *)
    DDI_ACTUAL_APPLICATION_RATE_OF_AMMONIUM : UINT := 437; (* 437 - Actual Application Rate of Ammonium *)
    DDI_MINIMUM_APPLICATION_RATE_OF_AMMONIUM : UINT := 438; (* 438 - Minimum Application Rate of Ammonium *)
    DDI_MAXIMUM_APPLICATION_RATE_OF_AMMONIUM : UINT := 439; (* 439 - Maximum Application Rate of Ammonium *)
    DDI_SETPOINT_APPLICATION_RATE_OF_PHOSPHOR : UINT := 440; (* 440 - Setpoint Application Rate of Phosphor *)
    DDI_ACTUAL_APPLICATION_RATE_OF_PHOSPHOR : UINT := 441; (* 441 - Actual Application Rate of Phosphor *)
    DDI_MINIMUM_APPLICATION_RATE_OF_PHOSPHOR : UINT := 442; (* 442 - Minimum Application Rate of Phosphor *)
    DDI_MAXIMUM_APPLICATION_RATE_OF_PHOSPHOR : UINT := 443; (* 443 - Maximum Application Rate of Phosphor *)
    DDI_SETPOINT_APPLICATION_RATE_OF_POTASSIUM : UINT := 444; (* 444 - Setpoint Application Rate of Potassium *)
    DDI_ACTUAL_APPLICATION_RATE_OF_POTASSIUM : UINT := 445; (* 445 - Actual Application Rate of Potassium *)
    DDI_MINIMUM_APPLICATION_RATE_OF_POTASSIUM : UINT := 446; (* 446 - Minimum Application Rate of Potassium *)
    DDI_MAXIMUM_APPLICATION_RATE_OF_POTASSIUM : UINT := 447; (* 447 - Maximum Application Rate of Potassium *)
    DDI_SETPOINT_APPLICATION_RATE_OF_DRY_MATTER : UINT := 448; (* 448 - Setpoint Application Rate of Dry Matter *)
    DDI_ACTUAL_APPLICATION_RATE_OF_DRY_MATTER : UINT := 449; (* 449 - Actual Application Rate of Dry Matter *)
    DDI_MINIMUM_APPLICATION_RATE_OF_DRY_MATTER : UINT := 450; (* 450 - Minimum Application Rate of Dry Matter *)
    DDI_MAXIMUM_APPLICATION_RATE_OF_DRY_MATTER : UINT := 451; (* 451 - Maximum Application Rate of Dry Matter *)
    DDI_LOADED_TOTAL_VOLUME : UINT := 452; (* 452 - Loaded Total Volume *)
    DDI_UNLOADED_TOTAL_VOLUME : UINT := 453; (* 453 - Unloaded Total Volume *)
    DDI_LIFETIME_LOADED_TOTAL_VOLUME : UINT := 454; (* 454 - Lifetime loaded Total Volume *)
    DDI_LIFETIME_UNLOADED_TOTAL_VOLUME : UINT := 455; (* 455 - Lifetime Unloaded Total Volume *)
    DDI_LAST_LOADED_VOLUME : UINT := 456; (* 456 - Last loaded Volume *)
    DDI_LAST_UNLOADED_VOLUME : UINT := 457; (* 457 - Last unloaded Volume *)
    DDI_LOADED_TOTAL_COUNT : UINT := 458; (* 458 - Loaded Total Count *)
    DDI_UNLOADED_TOTAL_COUNT : UINT := 459; (* 459 - Unloaded Total Count *)
    DDI_LIFETIME_LOADED_TOTAL_COUNT : UINT := 460; (* 460 - Lifetime Loaded Total Count *)
    DDI_LIFETIME_UNLOADED_TOTAL_COUNT : UINT := 461; (* 461 - Lifetime Unloaded Total Count *)
    DDI_LAST_LOADED_COUNT : UINT := 462; (* 462 - Last loaded Count *)
    DDI_LAST_UNLOADED_COUNT : UINT := 463; (* 463 - Last unloaded Count *)
    DDI_HAUL_COUNTER : UINT := 464; (* 464 - Haul Counter *)
    DDI_LIFETIME_HAUL_COUNTER : UINT := 465; (* 465 - Lifetime Haul Counter *)
    DDI_ACTUAL_RELATIVE_CONNECTOR_ANGLE : UINT := 466; (* 466 - Actual relative connector angle *)
    DDI_ACTUAL_PERCENTAGE_CONTENT : UINT := 467; (* 467 - Actual Percentage Content *)
    DDI_SOIL_SNOW_FROZEN_CONDTION : UINT := 468; (* 468 - Soil Snow/Frozen Condtion *)
    DDI_ESTIMATED_SOIL_WATER_CONDTION : UINT := 469; (* 469 - Estimated Soil Water Condtion *)
    DDI_SOIL_COMPACTION : UINT := 470; (* 470 - Soil Compaction *)
    DDI_SETPOINT_CULTURAL_PRACTICE : UINT := 471; (* 471 - Setpoint Cultural Practice *)
    DDI_SETPOINT_LENGTH_OF_CUT : UINT := 472; (* 472 - Setpoint Length of Cut *)
    DDI_MINIMUM_LENGTH_OF_CUT : UINT := 473; (* 473 - Minimum length of cut *)
    DDI_MAXIMUM_LENGTH_OF_CUT : UINT := 474; (* 474 - Maximum Length of Cut *)
    DDI_SETPOINT_BALE_HYDRAULIC_PRESSURE : UINT := 475; (* 475 - Setpoint Bale Hydraulic Pressure *)
    DDI_MINIMUM_BALE_HYDRAULIC_PRESSURE : UINT := 476; (* 476 - Minimum Bale Hydraulic Pressure *)
    DDI_MAXIMUM_BALE_HYDRAULIC_PRESSURE : UINT := 477; (* 477 - Maximum Bale Hydraulic Pressure *)
    DDI_SETPOINT_FLAKE_SIZE : UINT := 478; (* 478 - Setpoint Flake Size *)
    DDI_MINIMUM_FLAKE_SIZE : UINT := 479; (* 479 - Minimum Flake Size *)
    DDI_MAXIMUM_FLAKE_SIZE : UINT := 480; (* 480 - Maximum Flake Size *)
    DDI_SETPOINT_NUMBER_OF_SUBBALES : UINT := 481; (* 481 - Setpoint Number of Subbales *)
    DDI_LAST_BALE_NUMBER_OF_SUBBALES : UINT := 482; (* 482 - Last Bale Number of Subbales *)
    DDI_SETPOINT_ENGINE_SPEED : UINT := 483; (* 483 - Setpoint Engine Speed *)
    DDI_ACTUAL_ENGINE_SPEED : UINT := 484; (* 484 - Actual Engine Speed *)
    DDI_MINIMUM_ENGINE_SPEED : UINT := 485; (* 485 - Minimum Engine Speed *)
    DDI_MAXIMUM_ENGINE_SPEED : UINT := 486; (* 486 - Maximum Engine Speed *)
    DDI_DIESEL_EXHAUST_FLUID_TANK_PERCENTAGE_LEVEL : UINT := 488; (* 488 - Diesel Exhaust Fluid Tank Percentage Level *)
    DDI_MAXIMUM_DIESEL_EXHAUST_FLUID_TANK_CONTENT : UINT := 489; (* 489 - Maximum Diesel Exhaust Fluid Tank Content *)
    DDI_MAXIMUM_FUEL_TANK_CONTENT : UINT := 490; (* 490 - Maximum Fuel Tank Content *)
    DDI_FUEL_PERCENTAGE_LEVEL : UINT := 491; (* 491 - Fuel Percentage Level *)
    DDI_TOTAL_ENGINE_HOURS : UINT := 492; (* 492 - Total Engine Hours *)
    DDI_LIFETIME_ENGINE_HOURS : UINT := 493; (* 493 - Lifetime Engine Hours *)
    DDI_LAST_EVENT_PARTNER_ID_BYTE_1_4 : UINT := 494; (* 494 - Last Event Partner ID (Byte 1-4) *)
    DDI_LAST_EVENT_PARTNER_ID_BYTE_5_8 : UINT := 495; (* 495 - Last Event Partner ID (Byte 5-8) *)
    DDI_LAST_EVENT_PARTNER_ID_BYTE_9_12 : UINT := 496; (* 496 - Last Event Partner ID (Byte 9-12) *)
    DDI_LAST_EVENT_PARTNER_ID_BYTE_13_16 : UINT := 497; (* 497 - Last Event Partner ID (Byte 13-16) *)
    DDI_LAST_EVENT_PARTNER_ID_TYPE : UINT := 498; (* 498 - Last Event Partner ID Type *)
    DDI_LAST_EVENT_PARTNER_ID_MANUFACTURER_ID_CODE : UINT := 499; (* 499 - Last Event Partner ID Manufacturer ID Code *)
    DDI_LAST_EVENT_PARTNER_ID_DEVICE_CLASS : UINT := 500; (* 500 - Last Event Partner ID Device Class *)
    DDI_SETPOINT_ENGINE_TORQUE : UINT := 501; (* 501 - Setpoint Engine Torque *)
    DDI_ACTUAL_ENGINE_TORQUE : UINT := 502; (* 502 - Actual Engine Torque *)
    DDI_MINIMUM_ENGINE_TORQUE : UINT := 503; (* 503 - Minimum Engine Torque *)
    DDI_MAXIMUM_ENGINE_TORQUE : UINT := 504; (* 504 - Maximum Engine Torque *)
    DDI_TRAMLINE_CONTROL_LEVEL : UINT := 505; (* 505 - Tramline Control Level *)
    DDI_SETPOINT_TRAMLINE_CONTROL_LEVEL : UINT := 506; (* 506 - Setpoint Tramline Control Level *)
    DDI_TRAMLINE_SEQUENCE_NUMBER : UINT := 507; (* 507 - Tramline Sequence Number *)
    DDI_UNIQUE_A_B_GUIDANCE_REFERENCE_LINE_ID : UINT := 508; (* 508 - Unique A-B Guidance Reference Line ID *)
    DDI_ACTUAL_TRACK_NUMBER : UINT := 509; (* 509 - Actual Track Number *)
    DDI_TRACK_NUMBER_TO_THE_RIGHT : UINT := 510; (* 510 - Track Number to the right *)
    DDI_TRACK_NUMBER_TO_THE_LEFT : UINT := 511; (* 511 - Track Number to the left *)
    DDI_GUIDANCE_LINE_SWATH_WIDTH : UINT := 512; (* 512 - Guidance Line Swath Width *)
    DDI_GUIDANCE_LINE_DEVIATION : UINT := 513; (* 513 - Guidance Line Deviation *)
    DDI_GNSS_QUALITY : UINT := 514; (* 514 - GNSS Quality *)
    DDI_TRAMLINE_CONTROL_STATE : UINT := 515; (* 515 - Tramline Control State *)
    DDI_TRAMLINE_OVERDOSING_RATE : UINT := 516; (* 516 - Tramline Overdosing Rate *)
    DDI_SETPOINT_TRAMLINE_CONDENSED_WORK_STATE_1_16 : UINT := 517; (* 517 - Setpoint Tramline Condensed Work State *)
    DDI_ACTUAL_TRAMLINE_CONDENSED_WORK_STATE_1_16 : UINT := 518; (* 518 - Actual Tramline Condensed Work State (1-16) *)
    DDI_LAST_BALE_LIFETIME_COUNT : UINT := 519; (* 519 - Last Bale Lifetime Count *)
    DDI_ACTUAL_CANOPY_HEIGHT : UINT := 520; (* 520 - Actual Canopy Height *)
    DDI_GNSS_INSTALLATION_TYPE : UINT := 521; (* 521 - GNSS Installation Type *)
    DDI_TWINE_BALE_TOTAL_COUNT : UINT := 522; (* 522 - Twine Bale Total Count *)
    DDI_MESH_BALE_TOTAL_COUNT : UINT := 523; (* 523 - Mesh Bale Total Count *)
    DDI_LIFETIME_TWINE_BALE_TOTAL_COUNT : UINT := 524; (* 524 - Lifetime Twine Bale Total Count *)
    DDI_LIFETIME_MESH_BALE_TOTAL_COUNT : UINT := 525; (* 525 - Lifetime Mesh Bale Total Count *)
    DDI_ACTUAL_COOLING_FLUID_TEMPERATURE : UINT := 526; (* 526 - Actual Cooling Fluid Temperature *)
    DDI_LAST_BALE_CAPACITY : UINT := 528; (* 528 - Last Bale Capacity *)
    DDI_SETPOINT_TILLAGE_DISC_GANG_ANGLE : UINT := 529; (* 529 - Setpoint Tillage Disc Gang Angle *)
    DDI_ACTUAL_TILLAGE_DISC_GANG_ANGLE : UINT := 530; (* 530 - Actual Tillage Disc Gang Angle *)
    DDI_ACTUAL_APPLIED_PRESERVATIVE_PER_YIELD_MASS : UINT := 531; (* 531 - Actual Applied Preservative Per Yield Mass *)
    DDI_SETPOINT_APPLIED_PRESERVATIVE_PER_YIELD_MASS : UINT := 532; (* 532 - Setpoint Applied Preservative Per Yield *)
    DDI_DEFAULT_APPLIED_PRESERVATIVE_PER_YIELD_MASS : UINT := 533; (* 533 - Default Applied Preservative Per Yield *)
    DDI_MINIMUM_APPLIED_PRESERVATIVE_PER_YIELD_MASS : UINT := 534; (* 534 - Minimum Applied Preservative Per Yield *)
    DDI_MAXIMUM_APPLIED_PRESERVATIVE_PER_YIELD_MASS : UINT := 535; (* 535 - Maximum Applied Preservative Per Yield *)
    DDI_TOTAL_APPLIED_PRESERVATIVE : UINT := 536; (* 536 - Total Applied Preservative *)
    DDI_LIFETIME_APPLIED_PRESERVATIVE : UINT := 537; (* 537 - Lifetime Applied Preservative *)
    DDI_AVERAGE_APPLIED_PRESERVATIVE_PER_YIELD_MASS : UINT := 538; (* 538 - Average Applied Preservative Per Yield *)
    DDI_ACTUAL_PRESERVATIVE_TANK_VOLUME : UINT := 539; (* 539 - Actual Preservative Tank Volume *)
    DDI_ACTUAL_PRESERVATIVE_TANK_LEVEL : UINT := 540; (* 540 - Actual Preservative Tank Level *)
    DDI_ACTUAL_PTO_SPEED : UINT := 541; (* 541 - Actual PTO Speed *)
    DDI_SETPOINT_PTO_SPEED : UINT := 542; (* 542 - Setpoint PTO Speed *)
    DDI_DEFAULT_PTO_SPEED : UINT := 543; (* 543 - Default PTO Speed *)
    DDI_MINIMUM_PTO_SPEED : UINT := 544; (* 544 - Minimum PTO Speed *)
    DDI_MAXIMUM_PTO_SPEED : UINT := 545; (* 545 - Maximum PTO Speed *)
    DDI_LIFETIME_CHOPPING_ENGAGEMENT_TOTAL_TIME : UINT := 546; (* 546 - Lifetime Chopping Engagement Total Time *)
    DDI_SETPOINT_BALE_COMPRESSION_PLUNGER_LOAD_N : UINT := 547; (* 547 - Setpoint Bale Compression Plunger Load (N) *)
    DDI_ACTUAL_BALE_COMPRESSION_PLUNGER_LOAD_N : UINT := 548; (* 548 - Actual Bale Compression Plunger Load (N) *)
    DDI_LAST_BALE_AVERAGE_BALE_COMPRESSION_PLUNGER_LOAD_N : UINT := 549; (* 549 - Last Bale Average Bale Compression *)
    DDI_GROUND_COVER : UINT := 550; (* 550 - Ground Cover *)
    DDI_ACTUAL_PTO_TORQUE : UINT := 551; (* 551 - Actual PTO Torque *)
    DDI_SETPOINT_PTO_TORQUE : UINT := 552; (* 552 - Setpoint PTO Torque *)
    DDI_DEFAULT_PTO_TORQUE : UINT := 553; (* 553 - Default PTO Torque *)
    DDI_MINIMUM_PTO_TORQUE : UINT := 554; (* 554 - Minimum PTO Torque *)
    DDI_MAXIMUM_PTO_TORQUE : UINT := 555; (* 555 - Maximum PTO Torque *)
    DDI_PRESENT_WEATHER_CONDITIONS : UINT := 556; (* 556 - Present Weather Conditions *)
    DDI_SETPOINT_ELECTRICAL_CURRENT : UINT := 557; (* 557 - Setpoint Electrical Current *)
    DDI_ACTUAL_ELECTRICAL_CURRENT : UINT := 558; (* 558 - Actual Electrical Current *)
    DDI_MINIMUM_ELECTRICAL_CURRENT : UINT := 559; (* 559 - Minimum Electrical Current *)
    DDI_MAXIMUM_ELECTRICAL_CURRENT : UINT := 560; (* 560 - Maximum Electrical Current *)
    DDI_DEFAULT_ELECTRICAL_CURRENT : UINT := 561; (* 561 - Default Electrical Current *)
    DDI_SETPOINT_VOLTAGE : UINT := 562; (* 562 - Setpoint Voltage *)
    DDI_DEFAULT_VOLTAGE : UINT := 563; (* 563 - Default Voltage *)
    DDI_ACTUAL_VOLTAGE : UINT := 564; (* 564 - Actual Voltage *)
    DDI_MINIMUM_VOLTAGE : UINT := 565; (* 565 - Minimum Voltage *)
    DDI_MAXIMUM_VOLTAGE : UINT := 566; (* 566 - Maximum Voltage *)
    DDI_ACTUAL_ELECTRICAL_RESISTANCE : UINT := 567; (* 567 - Actual Electrical Resistance *)
    DDI_SETPOINT_ELECTRICAL_POWER : UINT := 568; (* 568 - Setpoint Electrical Power *)
    DDI_ACTUAL_ELECTRICAL_POWER : UINT := 569; (* 569 - Actual Electrical Power *)
    DDI_DEFAULT_ELECTRICAL_POWER : UINT := 570; (* 570 - Default Electrical Power *)
    DDI_MAXIMUM_ELECTRICAL_POWER : UINT := 571; (* 571 - Maximum Electrical Power *)
    DDI_MINIMUM_ELECTRICAL_POWER : UINT := 572; (* 572 - Minimum Electrical Power *)
    DDI_TOTAL_ELECTRICAL_ENERGY : UINT := 573; (* 573 - Total Electrical Energy *)
    DDI_SETPOINT_ELECTRICAL_ENERGY_PER_AREA_APPLICATION_RATE : UINT := 574; (* 574 - Setpoint Electrical Energy per *)
    DDI_ACTUAL_ELECTRICAL_ENERGY_PER_AREA_APPLICATION_RATE : UINT := 575; (* 575 - Actual Electrical Energy per Area *)
    DDI_MAXIMUM_ELECTRICAL_ENERGY_PER_AREA_APPLICATION_RATE : UINT := 576; (* 576 - Maximum Electrical Energy per *)
    DDI_MINIMUM_ELECTRICAL_ENERGY_PER_AREA_APPLICATION_RATE : UINT := 577; (* 577 - Minimum Electrical Energy per *)
    DDI_SETPOINT_TEMPERATURE : UINT := 578; (* 578 - Setpoint Temperature *)
    DDI_ACTUAL_TEMPERATURE : UINT := 579; (* 579 - Actual Temperature *)
    DDI_MINIMUM_TEMPERATURE : UINT := 580; (* 580 - Minimum Temperature *)
    DDI_MAXIMUM_TEMPERATURE : UINT := 581; (* 581 - Maximum Temperature *)
    DDI_DEFAULT_TEMPERATURE : UINT := 582; (* 582 - Default Temperature *)
    DDI_SETPOINT_FREQUENCY : UINT := 583; (* 583 - Setpoint Frequency *)
    DDI_ACTUAL_FREQUENCY : UINT := 584; (* 584 - Actual Frequency *)
    DDI_MINIMUM_FREQUENCY : UINT := 585; (* 585 - Minimum Frequency *)
    DDI_MAXIMUM_FREQUENCY : UINT := 586; (* 586 - Maximum Frequency *)
    DDI_PREVIOUS_RAINFALL : UINT := 587; (* 587 - Previous Rainfall *)
    DDI_SETPOINT_VOLUME_PER_AREA_APPLICATION_RATE_BIG : UINT := 588; (* 588 - Setpoint Volume Per Area *)
    DDI_ACTUAL_VOLUME_PER_AREA_APPLICATION_RATE_BIG : UINT := 589; (* 589 - Actual Volume Per Area Application *)
    DDI_MINIMUM_VOLUME_PER_AREA_APPLICATION_RATE_BIG : UINT := 590; (* 590 - Minimum Volume Per Area Application *)
    DDI_MAXIMUM_VOLUME_PER_AREA_APPLICATION_RATE_BIG : UINT := 591; (* 591 - Maximum Volume Per Area Application *)
    DDI_DEFAULT_VOLUME_PER_AREA_APPLICATION_RATE_BIG : UINT := 592; (* 592 - Default Volume Per Area Application *)
    DDI_TRACTION_TYPE : UINT := 593; (* 593 - Traction Type *)
    DDI_STEERING_TYPE : UINT := 594; (* 594 - Steering Type *)
    DDI_MACHINE_MODE : UINT := 595; (* 595 - Machine Mode *)
    DDI_CARGO_AREA_COVER_STATE : UINT := 596; (* 596 - Cargo Area Cover State *)
    DDI_TOTAL_DISTANCE : UINT := 597; (* 597 - Total Distance *)
    DDI_LIFETIME_TOTAL_DISTANCE : UINT := 598; (* 598 - Lifetime Total Distance *)
    DDI_TOTAL_DISTANCE_FIELD : UINT := 599; (* 599 - Total Distance Field *)
    DDI_LIFETIME_TOTAL_DISTANCE_FIELD : UINT := 600; (* 600 - Lifetime Total Distance Field *)
    DDI_TOTAL_DISTANCE_STREET : UINT := 601; (* 601 - Total Distance Street *)
    DDI_LIFETIME_TOTAL_DISTANCE_STREET : UINT := 602; (* 602 - Lifetime Total Distance Street *)
    DDI_ACTUAL_TRAMLINE_CONDENSED_WORK_STATE_17_32 : UINT := 603; (* 603 - Actual Tramline Condensed Work State *)
    DDI_ACTUAL_TRAMLINE_CONDENSED_WORK_STATE_33_48 : UINT := 604; (* 604 - Actual Tramline Condensed Work State *)
    DDI_ACTUAL_TRAMLINE_CONDENSED_WORK_STATE_49_64 : UINT := 605; (* 605 - Actual Tramline Condensed Work State *)
    DDI_ACTUAL_TRAMLINE_CONDENSED_WORK_STATE_65_80 : UINT := 606; (* 606 - Actual Tramline Condensed Work State *)
    DDI_ACTUAL_TRAMLINE_CONDENSED_WORK_STATE_81_96 : UINT := 607; (* 607 - Actual Tramline Condensed Work State *)
    DDI_ACTUAL_TRAMLINE_CONDENSED_WORK_STATE_97_112 : UINT := 608; (* 608 - Actual Tramline Condensed Work State *)
    DDI_ACTUAL_TRAMLINE_CONDENSED_WORK_STATE_113_128 : UINT := 609; (* 609 - Actual Tramline Condensed Work State *)
    DDI_ACTUAL_TRAMLINE_CONDENSED_WORK_STATE_129_144 : UINT := 610; (* 610 - Actual Tramline Condensed Work State *)
    DDI_ACTUAL_TRAMLINE_CONDENSED_WORK_STATE_145_160 : UINT := 611; (* 611 - Actual Tramline Condensed Work State *)
    DDI_ACTUAL_TRAMLINE_CONDENSED_WORK_STATE_161_176 : UINT := 612; (* 612 - Actual Tramline Condensed Work State *)
    DDI_ACTUAL_TRAMLINE_CONDENSED_WORK_STATE_177_192 : UINT := 613; (* 613 - Actual Tramline Condensed Work State *)
    DDI_ACTUAL_TRAMLINE_CONDENSED_WORK_STATE_193_208 : UINT := 614; (* 614 - Actual Tramline Condensed Work State *)
    DDI_ACTUAL_TRAMLINE_CONDENSED_WORK_STATE_209_224 : UINT := 615; (* 615 - Actual Tramline Condensed Work State *)
    DDI_ACTUAL_TRAMLINE_CONDENSED_WORK_STATE_225_240 : UINT := 616; (* 616 - Actual Tramline Condensed Work State *)
    DDI_ACTUAL_TRAMLINE_CONDENSED_WORK_STATE_241_256 : UINT := 617; (* 617 - Actual Tramline Condensed Work State *)
    DDI_SETPOINT_TRAMLINE_CONDENSED_WORK_STATE_17_32 : UINT := 618; (* 618 - Setpoint Tramline Condensed Work State *)
    DDI_SETPOINT_TRAMLINE_CONDENSED_WORK_STATE_33_48 : UINT := 619; (* 619 - Setpoint Tramline Condensed Work State *)
    DDI_SETPOINT_TRAMLINE_CONDENSED_WORK_STATE_49_64 : UINT := 620; (* 620 - Setpoint Tramline Condensed Work State *)
    DDI_SETPOINT_TRAMLINE_CONDENSED_WORK_STATE_65_80 : UINT := 621; (* 621 - Setpoint Tramline Condensed Work State *)
    DDI_SETPOINT_TRAMLINE_CONDENSED_WORK_STATE_81_96 : UINT := 622; (* 622 - Setpoint Tramline Condensed Work State *)
    DDI_SETPOINT_TRAMLINE_CONDENSED_WORK_STATE_97_112 : UINT := 623; (* 623 - Setpoint Tramline Condensed Work State *)
    DDI_SETPOINT_TRAMLINE_CONDENSED_WORK_STATE_113_128 : UINT := 624; (* 624 - Setpoint Tramline Condensed Work State *)
    DDI_SETPOINT_TRAMLINE_CONDENSED_WORK_STATE_129_144 : UINT := 625; (* 625 - Setpoint Tramline Condensed Work State *)
    DDI_SETPOINT_TRAMLINE_CONDENSED_WORK_STATE_145_160 : UINT := 626; (* 626 - Setpoint Tramline Condensed Work State *)
    DDI_SETPOINT_TRAMLINE_CONDENSED_WORK_STATE_161_176 : UINT := 627; (* 627 - Setpoint Tramline Condensed Work State *)
    DDI_SETPOINT_TRAMLINE_CONDENSED_WORK_STATE_177_192 : UINT := 628; (* 628 - Setpoint Tramline Condensed Work State *)
    DDI_SETPOINT_TRAMLINE_CONDENSED_WORK_STATE_193_208 : UINT := 629; (* 629 - Setpoint Tramline Condensed Work State *)
    DDI_SETPOINT_TRAMLINE_CONDENSED_WORK_STATE_209_224 : UINT := 630; (* 630 - Setpoint Tramline Condensed Work State *)
    DDI_SETPOINT_TRAMLINE_CONDENSED_WORK_STATE_225_240 : UINT := 631; (* 631 - Setpoint Tramline Condensed Work State *)
    DDI_SETPOINT_TRAMLINE_CONDENSED_WORK_STATE_241_256 : UINT := 632; (* 632 - Setpoint Tramline Condensed Work State *)
    DDI_SETPOINT_VOLUME_PER_DISTANCE_APPLICATION_RATE : UINT := 633; (* 633 - Setpoint Volume per distance *)
    DDI_ACTUAL_VOLUME_PER_DISTANCE_APPLICATION_RATE : UINT := 634; (* 634 - Actual Volume per distance Application *)
    DDI_DEFAULT_VOLUME_PER_DISTANCE_APPLICATION_RATE : UINT := 635; (* 635 - Default Volume per distance Application *)
    DDI_MINIMUM_VOLUME_PER_DISTANCE_APPLICATION_RATE : UINT := 636; (* 636 - Minimum Volume per distance Application *)
    DDI_MAXIMUM_VOLUME_PER_DISTANCE_APPLICATION_RATE : UINT := 637; (* 637 - Maximum Volume per distance Application *)
    DDI_SETPOINT_TIRE_PRESSURE : UINT := 638; (* 638 - Setpoint Tire Pressure *)
    DDI_ACTUAL_TIRE_PRESSURE : UINT := 639; (* 639 - Actual Tire Pressure *)
    DDI_DEFAULT_TIRE_PRESSURE : UINT := 640; (* 640 - Default Tire Pressure *)
    DDI_MINIMUM_TIRE_PRESSURE : UINT := 641; (* 641 - Minimum Tire Pressure *)
    DDI_MAXIMUM_TIRE_PRESSURE : UINT := 642; (* 642 - Maximum Tire Pressure *)
    DDI_ACTUAL_TIRE_TEMPERATURE : UINT := 643; (* 643 - Actual Tire Temperature *)
    DDI_BINDING_METHOD : UINT := 644; (* 644 - Binding Method *)
    DDI_LAST_BALE_NUMBER_OF_KNIVES : UINT := 645; (* 645 - Last Bale Number of Knives *)
    DDI_LAST_BALE_TWINE_CONSUMPTION : UINT := 646; (* 646 - Last Bale Twine Consumption *)
    DDI_LAST_BALE_MESH_CONSUMPTION : UINT := 647; (* 647 - Last Bale Mesh Consumption *)
    DDI_LAST_BALE_FILM_CONSUMPTION : UINT := 648; (* 648 - Last Bale Film Consumption *)
    DDI_LAST_BALE_FILM_STRETCHING : UINT := 649; (* 649 - Last Bale Film Stretching *)
    DDI_LAST_BALE_WRAPPING_FILM_WIDTH : UINT := 650; (* 650 - Last Bale Wrapping Film Width *)
    DDI_LAST_BALE_WRAPPING_FILM_CONSUMPTION : UINT := 651; (* 651 - Last Bale Wrapping Film Consumption *)
    DDI_LAST_BALE_WRAPPING_FILM_STRETCHING : UINT := 652; (* 652 - Last Bale Wrapping Film Stretching *)
    DDI_LAST_BALE_WRAPPING_FILM_OVERLAP_PERCENTAGE : UINT := 653; (* 653 - Last Bale Wrapping Film Overlap Percentage *)
    DDI_LAST_BALE_WRAPPING_FILM_LAYERS : UINT := 654; (* 654 - Last Bale Wrapping Film Layers *)
    DDI_ELECTRICAL_APPARENT_SOIL_CONDUCTIVITY : UINT := 655; (* 655 - Electrical Apparent Soil Conductivity *)
    DDI_SC_ACTUAL_TURN_ON_TIME : UINT := 656; (* 656 - SC Actual Turn On Time *)
    DDI_SC_ACTUAL_TURN_OFF_TIME : UINT := 657; (* 657 - SC Actual Turn Off Time *)
    DDI_MAXIMUM_DROPLET_SIZE : UINT := 32768; (* 32768 - Maximum Droplet Size *)
    DDI_MINIMUM_DROPLET_SIZE : UINT := 36864; (* 36864 - Minimum Droplet Size *)
    DDI_DEFAULT_DROPLET_SIZE : UINT := 40960; (* 40960 - Default Droplet Size *)
    DDI_ACTUAL_DROPLET_SIZE : UINT := 45056; (* 45056 - Actual Droplet Size *)
    DDI_SETPOINT_DROPLET_SIZE : UINT := 49152; (* 49152 - Setpoint Droplet Size *)
    DDI_PGN_BASED_DATA : UINT := 57342; (* 57342 - PGN Based Data *)
    DDI_REQUEST_DEFAULT_PROCESS_DATA : UINT := 57343; (* 57343 - Request Default Process Data *)
    DDI_PROPRIETARY_DDI_RANGE_START : UINT := 57344; (* 57344 - Proprietary DDI Range START *)
    DDI_PROPRIETARY_DDI_RANGE_END : UINT := 65534; (* 65534 - Proprietary DDI Range END *)
    DDI_RESERVED : UINT := 65535; (* 65535 - Reserved *)
  END_VAR
END_GLOBALCONSTANTS
